// TIA Portal V20 export
TYPE "typeCmInterfaceBrakeTest"
// stored: Access Published, Namespace Unit1.Em5
   STRUCT
      magazine : "LER_typeBrakeTestEmInterface";
   END_STRUCT;
END_TYPE
